PROGRAM MsgControl
VAR_INPUT
	TransmitEnable 				: BOOL;
	nConnectionIndex			: UDINT	:= 1;
END_VAR
VAR
	MsgID						: DINT;			// TCP/IP Message ID as per Communication protocol defined in FA 
	DeviceID					: STRING(5);	// TCP/IP Device ID as per Communication protocol defined in FA 
	BarCode						: STRING(20);	// TCP/IP Load ID (Bar Code) as per Communication protocol defined in FA
	BarCodeNoSpace				: STRING(20);	// TCP/IP Load ID (Bar Code) as per Communication protocol defined in FA stripped of spaces  
	Destination					: DINT;			// TCP/IP Destination as per Communication protocol defined in FA
	DefDestination				: DINT;			// TCP/IP Default Destination as per Communication protocol defined in FA
	Status						: BYTE;				// 
	Msg_EquipStatArry			: ARRAY[1..7] OF ST_Msg_EquipStat;
	nSystemStatusIndex 			: DINT; 	// Index used for Processing the system status array
	nTempOperState 				: DINT;	//Capture the Temporary Operating State of the Equipment for comparison
	nEquipStatusIndex			: DINT;	//Index used for adding items to the MSG_EquipStatArray
	StrStartPos					: INT;
	StrEndPos					: INT;
	MsgString					: STRING(55);
	RawMsgArray					: ARRAY[1..10] OF T_MaxString;	// Capture the last Raw messages for troubleshooting
	RawMsgLenArray				: ARRAY[1..10] OF INT;			// Capture the last  Raw message lengths for troubleshooting
	RawMsgStartPosArray			: ARRAY[1..10] OF INT;			// Capture the last  Raw message start positions for troubleshooting
	RawMsgEndPosArray			: ARRAY[1..10] OF INT;			// Capture the last  Raw message end positions for troubleshooting
	MsgArray					: ARRAY[1..10] OF STRING(55);		// Capture the last 10 messages that have been stripped from the starting character  for troubleshooting
	Blank_Msg_ConveyorStatArry	: ARRAY [1..7] OF ST_Msg_EquipStat := [7((Status := 99))];

	i 							: INT;
	j							: INT;
	
	RxCounter_Old				: UDINT;
	TxCounter_Old				: UDINT;
	TransmitMsgBuffer			: ARRAY [1..TransmitMsgBuffer_Size] OF STRING(55);	// Buffer to hold transmit messages
	TransmitMsgBuffer_Index		: INT :=	1;		// Index to the Buffer
	TransmitMsgStatus			: INT;			
	SendingMsg_Index			: INT :=	1;		// Index to send message
	
	ItemTransport				: ST_Item;		// Output Item Update with destination from ARUP Host (Send to Sorter PLC)
	BlankItem					: ST_Item := (ID := '', UniqueID := 0
													, Destination := 0
													, Status := E_StatusCode.No_Status
													, ExtStatus := E_StatusCode.No_Status
													, DeviceID := ''
													, MessageType := E_MessageIds.NoMessage_00);

	ReadBCRID_S2140_01_Old			: UDINT;		// Bar Code watch variable
	ReadBCRID_S2141_01_Old			: UDINT;		// Bar Code watch variable
	ReadBCRID_S2150_01_Old			: UDINT;		// Bar Code watch variable	
	ReadBCRID_S3080_01_Old			: UDINT;		// Bar Code watch variable
			
	TransmittedArray			: ARRAY[0..10] OF STRING(55);
	x							: DINT;
	y							: INT;
	
	SpacePosition				: INT;
	
	fb_CheckStopRegister		: FB_ManageCodes;	// Used to test for a specific Stop Code to report to the Host
	bOverHeight					: BOOL; 	// Detect OverHeight to report to the Host
	st_UpdateMessageToSend		: ST_Item;			// Message to Send to Host

	fb_SorterUpdateBuffer			: FB_ItemBuffer;	// Function to Process the SorterUpdateBuffer

	fb_SorterTransportBuffer_P2140	: FB_ItemBuffer;	// Function to Process the SorterTransportBuffer
	fb_SorterTransportBuffer_P2150	: FB_ItemBuffer;	// Function to Process the SorterTransportBuffer

	sMessage	:	STRING;
	
END_VAR

VAR CONSTANT
	SEND_ARRIVAL			:	INT := 5;
	SEND_LOCATION			:	INT := 7;
	TransmitMsgBuffer_Size	:	INT :=	25;		// Number of Messages to hold in buffer
END_VAR

// Create instances of Buffer Processing Functions to initialize the buffers and data
fb_SorterUpdateBuffer.Master := FALSE;
fb_SorterTransportBuffer_P2140.Master := TRUE;
fb_SorterTransportBuffer_P2150.Master := TRUE;

// Activate or de-activate logging
fb_SorterUpdateBuffer.LogEntries := .nItemBufferLogEnable.UPDATE OR .nItemBufferLogEnableP2150.UPDATE OR .nItemBufferLogEnableP2150.UPDATE;
fb_SorterTransportBuffer_P2140.LogEntries := .nItemBufferLogEnable.TRANSPORT OR .nItemBufferLogEnableP2140.TRANSPORT;
fb_SorterTransportBuffer_P2150.LogEntries := .nItemBufferLogEnable.TRANSPORT OR .nItemBufferLogEnableP2150.TRANSPORT;

// Setup Buffer names for Logging purposes
fb_SorterUpdateBuffer.Name := 'SYS UPDATE';
fb_SorterTransportBuffer_P2140.Name := 'P2140 SYS TRANSPORT';
fb_SorterTransportBuffer_P2150.Name := 'P2150 SYS TRANSPORT';

fb_SorterUpdateBuffer(st_BufferData := st_SorterUpdateBuffer
					, st_BufferFdbkIn := st_UpdateFdbkOut
					, st_BufferFdbkOut => st_UpdateFdbkIn);
fb_SorterTransportBuffer_P2140(st_BufferData := st_SorterTransportBuffer_P2140
					, st_BufferFdbkIn := st_TransportFdbkIn_P2140
					, st_BufferFdbkOut => st_TransportFdbkOut_P2140);
fb_SorterTransportBuffer_P2150(st_BufferData := st_SorterTransportBuffer_P2150
					, st_BufferFdbkIn := st_TransportFdbkIn_P2150
					, st_BufferFdbkOut => st_TransportFdbkOut_P2150);

(* -------------------- On Receive Message Process the data -------------------- *)
IF RxCounter_Old <> ServerControl.fbServer.aApplications[nConnectionIndex].RxCounter  THEN
	ItemTransport := BlankItem; // Clear the ItemTransport each pass to capture only new transport commands
	RECEIVE();
	// Test the DeviceID and route the Transport accordingly
	//	If there is only one possible DeviceID, this IF statement can be removed, but the fb_(TransportBuffer).AddItem call still has to be made
	//	Also, the default destination needs to be passed per DeviceID
	IF DeviceID = Sorter.st_Sorter_P2140Cfg.EquipID THEN
		// Added temporaily because code change needed on ARUP side 
			IF ItemTransport.Destination =0 THEN
			ItemTransport.Destination := 1;
			ELSIF ItemTransport.Destination =1 THEN
				ItemTransport.Destination := 2;
			END_IF
			// End addition	
		fb_SorterTransportBuffer_P2140.AddItem(st_ItemToAdd := ItemTransport);
		P2140_DefaultDestination := DefDestination;
	END_IF
	IF DeviceID = Sorter.st_Sorter_P2150Cfg.EquipID THEN
		fb_SorterTransportBuffer_P2150.AddItem(st_ItemToAdd := ItemTransport);
		P2150_DefaultDestination := DefDestination;
	END_IF

	RxCounter_Old := ServerControl.fbServer.aApplications[nConnectionIndex].RxCounter;
END_IF

(* -------------------- Transmit Messages if any are waiting in the buffer --------------------- *)
IF SendingMsg_Index <> TransmitMsgBuffer_Index THEN
	TRANSMIT(TransmitEnable:= TRUE);
END_IF

(* -------------------- Watch Bar code readers and send message when load is read -------------------- *)
(* ----- BCR_S2140_01: P2140 Divert  ----- *)	
ReadBCRID_S2140_01_Old := BarCodeMessage(cDatamanReader := BarCodeReaders.BCR_S2140_01
									, nOldCount := ReadBCRID_S2140_01_Old
									, nMessageToSend := SEND_ARRIVAL);
(* ----- BCR_S2141_01: P2143 Induct Confirm ----- *)	
ReadBCRID_S2141_01_Old := BarCodeMessage(cDatamanReader := BarCodeReaders.BCR_S2141_01
									, nOldCount := ReadBCRID_S2141_01_Old
									, nMessageToSend := SEND_LOCATION);
(* ----- BCR_S2150_01: P2150 Sorter ----- *)	
ReadBCRID_S2150_01_Old := BarCodeMessage(cDatamanReader := BarCodeReaders.BCR_S2150_01
									, nOldCount := ReadBCRID_S2150_01_Old
									, nMessageToSend := SEND_ARRIVAL);
(* ----- BCR_S3080_01: P3080 Lane Confirm ----- *)	
ReadBCRID_S3080_01_Old := BarCodeMessage(cDatamanReader := BarCodeReaders.BCR_S3080_01
									, nOldCount := ReadBCRID_S3080_01_Old
									, nMessageToSend := SEND_LOCATION);


(* -------------------- Watch Sorter and Device Status and transmit on change -------------------- *)
// Transmit On update from Sorter
// Detect a new message to process when the in and out pointer values disagree
IF st_SorterUpdateBuffer.nInPointer <> fb_SorterUpdateBuffer.OutPointer THEN
	// Pull the next message out of the buffer
	fb_SorterUpdateBuffer.RemoveItem(st_ItemToReturn => st_UpdateMessageToSend);
	CASE st_UpdateMessageToSend.MessageType OF

		E_MessageIds.TransportResponse_25:			// Response to a Transport Command

			CASE st_UpdateMessageToSend.Status OF
				E_StatusCode.Assign_Accepted:		// Assignment Accepted
					TransmitMsgStatus := E_TransportResponse.Accepted; 
				E_StatusCode.Assign_Full:			// Assigned Lane Unavailable
					TransmitMsgStatus := E_TransportResponse.DivertLaneUnavailable; 
				E_StatusCode.Assign_NotFound:		// Assigned Load ID Not Found
					TransmitMsgStatus := E_TransportResponse.LoadIdNotFound; 
				E_StatusCode.Assign_NotInducted:	// Assigned Load Not Inducted
					TransmitMsgStatus := E_TransportResponse.NextLoadReady; 
				E_StatusCode.Diverting:	// Assigned Load already Inducting
					TransmitMsgStatus := E_TransportResponse.LateInduction; 
			ELSE
				TransmitMsgStatus := E_TransportResponse.UnknownFailure; // Capture any other failures
				IF nMessageLogEnable.TransportResponse_25 THEN
					sMessage := CONCAT(' Item: ', st_UpdateMessageToSend.ID);
					sMessage := CONCAT(sMessage,' Destination: ');
					sMessage := CONCAT(sMessage, DINT_TO_STRING(st_UpdateMessageToSend.Destination));
					sMessage := CONCAT(sMessage,' TR Status: ');
					sMessage := CONCAT(sMessage, DINT_TO_STRING(st_UpdateMessageToSend.Status));
					// Write to the Error List
					ADSLOGSTR( msgCtrlMask := ADSLOG_MSGTYPE_HINT OR ADSLOG_MSGTYPE_LOG
						, msgFmtStr := 'Unhandled Transport Response Status: %s'
						, strArg := sMessage);
				END_IF
			END_CASE
			TransmitMsgBuffer[TransmitMsgBuffer_Index] := TransportResponse(Device := st_UpdateMessageToSend.DeviceID
																			, Barcode := st_UpdateMessageToSend.ID
																			, Status := TransmitMsgStatus);
			TransmitMsgBuffer_Index := IncIndex(TransmitMsgBuffer_Index,1,TransmitMsgBuffer_Size);

		E_MessageIds.TransportComplete_26:			// Indication of the final disposition of a transported item

			CASE st_UpdateMessageToSend.Status OF
				E_StatusCode.Divert_Success:		// Divert Success Message
					TransmitMsgStatus := E_TransportComplete.Success; 
				E_StatusCode.Divert_Complete:		// Divert Success Message
					TransmitMsgStatus := E_TransportComplete.Success; 
			ELSE 									// Catch all other failures
				TransmitMsgStatus := E_TransportComplete.Faulted; 
			END_CASE			
			CASE st_UpdateMessageToSend.ExtStatus OF
				E_StatusCode.Divert_Full:			// Divert Full/Unavailable
					TransmitMsgStatus := E_TransportComplete.Unavailable; 
				E_StatusCode.Divert_Offline:		// Divert Offline
					TransmitMsgStatus := E_TransportComplete.Offline; 
				E_StatusCode.Divert_Missed:		// Divert Missed
					TransmitMsgStatus := E_TransportComplete.Passed; 
				E_StatusCode.Divert_Recirculated:		// Divert Missed
					TransmitMsgStatus := E_TransportComplete.Success; 
			END_CASE			
			TransmitMsgBuffer[TransmitMsgBuffer_Index] := TransportComplete(Device:= st_UpdateMessageToSend.DeviceID
																			, BarCode:= st_UpdateMessageToSend.ID
																			, Dest:= DINT_TO_INT(st_UpdateMessageToSend.Destination)
																			, Status:= TransmitMsgStatus ); 
			TransmitMsgBuffer_Index := IncIndex(TransmitMsgBuffer_Index,1,TransmitMsgBuffer_Size);

	END_CASE
END_IF

// Transmit on Device Status Change
//DeviceStatus();1


(* -------------------- Reset The Transmit Triger after the message is succesfully added to the buffer ------------------- *)
IF ((ServerControl.fbServer.aApplications[nConnectionIndex].bTransmitTrigger = TRUE) OR ServerControl.TransmitTrigger = TRUE)  AND (TxCounter_Old <> ServerControl.fbServer.aApplications[nConnectionIndex].TxCounter) THEN
	ServerControl.TransmitTrigger := FALSE;
	TRANSMIT(TransmitEnable:= FALSE);
	TxCounter_Old := ServerControl.fbServer.aApplications[nConnectionIndex].TxCounter;
END_IF

METHOD PRIVATE Arrival : STRING(55)
VAR_INPUT
	Device :	STRING(5);		// Device Label per communication standard
	BarCode:	STRING(30);		// Barcode from barcode reader
	DefDest:	INT;		// Default destination
END_VAR
VAR
	String1: STRING(55);
	BC_Len: INT;
	x: INT;
	String_DefDest: STRING(2);
	y: INT;
	Device_Len: INT;
	i: INT;
END_VAR
(* Message from communication Spec:
	[STX (0x02h)][23][Device ID (5 CHR)][Barcode (20 CHR)][Default Dest (2 CHR)][Blank (22 CHR)][ETX 0x03h)]
*)

// Start Message with header
String1 := '$0223';

// Check Device for length and Pad with spaces if needed
Device_Len := LEN(Device);
IF Device_Len = 5 THEN
	String1 := CONCAT(STRING1, Device);
ELSIF Device_Len < 5 THEN
	String1 := CONCAT(STRING1, Device);
	FOR i := 1 TO (5-Device_Len) DO
		String1 := CONCAT(String1,' ');
	END_FOR
ELSE
	String1 := CONCAT(String1, 'XXXXX');
END_IF

// Check Barcode for length and Pad with spaces if needed
BC_Len := LEN(BARCODE);
IF BC_Len <20 THEN
	String1 := CONCAT(STRING1, BarCode);
	FOR x := 1 TO (20-BC_Len) DO
		String1 := CONCAT(String1,' ');
	END_FOR
ELSIF BC_Len = 20 THEN
	String1 := CONCAT(STRING1, BarCode);
ELSE 
	String1 := CONCAT(STRING1, RIGHT(BarCode,20));	
END_IF

// Check Default Destination for length and Pad with spaces if needed
String_DefDest := INT_TO_STRING(DefDest);
IF DefDest < 10 THEN
	String1 := CONCAT(String1,'0');
	String1 := CONCAT(String1, String_DefDest);
ELSIF (DefDest >= 10) AND (DefDest < 100) THEN
	String1 := CONCAT(String1, String_DefDest);
ELSE
	String1 := CONCAT(String1, 'XX');
END_IF	

// Pad with spaces
FOR y := 1 TO 22 DO
	String1 := CONCAT(String1,' ');
END_FOR

// Add ending Character
String1 := CONCAT(String1,'$03');
	
Arrival := String1;
END_METHOD

METHOD PRIVATE BarCodeMessage : UDINT
VAR_INPUT
	cDatamanReader	: CognexDataMan260;
//	sLocation		:	STRING(5);
	nOldCount		:	UDINT;
	nMessageToSend	: 	INT;
END_VAR
IF nOldCount <> cDatamanReader.GoodreadCount THEN
	// Send location update message to host
	CASE nMessageToSend OF
		SEND_ARRIVAL:	TransmitMsgBuffer[TransmitMsgBuffer_Index] := Arrival(cDatamanReader.In_EquipID, cDatamanReader.Out_ReadString,00);
		SEND_LOCATION: TransmitMsgBuffer[TransmitMsgBuffer_Index] := LocationUpdate(cDatamanReader.In_EquipID, cDatamanReader.Out_ReadString,00);
	END_CASE
	TransmitMsgBuffer_Index := IncIndex(TransmitMsgBuffer_Index,1,TransmitMsgBuffer_Size);
	BarCodeMessage := cDatamanReader.GoodreadCount;
ELSE
	BarCodeMessage := nOldCount;
END_IF
END_METHOD

METHOD PRIVATE CustomMessage : UDINT
VAR_INPUT
	EquipID			: 	STRING(5);
	Barcode			:	STRING(30);
	nReadCount		:	UDINT;
	nOldCount		:	UDINT;
	nMessageToSend	: 	INT;
END_VAR
IF nOldCount <> nReadCount THEN
	// Send location update message to host
	CASE nMessageToSend OF
		SEND_ARRIVAL:	TransmitMsgBuffer[TransmitMsgBuffer_Index] := Arrival(EquipID, BarCode,00);
		SEND_LOCATION: TransmitMsgBuffer[TransmitMsgBuffer_Index] := LocationUpdate(EquipID, BarCode,00);
	END_CASE
	TransmitMsgBuffer_Index := IncIndex(TransmitMsgBuffer_Index,1,TransmitMsgBuffer_Size);
	CustomMessage := nReadCount;
ELSE
	CustomMessage := nOldCount;
END_IF
END_METHOD

ACTION DeviceStatus:
(*
	
	Local Data items used for Equipment status processing
	Msg_EquipStatArry:	ARRAY[1..7] OF ST_Msg_EquipStat;
	nSystemStatusIndex : INT; 	// Index used for Processing the system status array
	nEquipStatusIndex: INT;	//Index used for adding items to the MSG_EquipStatArray
	nTempOperState : DINT;	//Capture the Temporary Operating State of the Equipment for comparison
	
	GVL_EquipmentArray items used for Equipment Status processing
	// System Equipment
	SystemEquip_Count : INT; //Count of Equipment to Process in System PLC
	SystemEquipStatusArray : ARRAY[1..EQUIP_COUNT_MAX] OF ST_StateCntrlSts; //Array of Equipment Status Current
	SystemEquipStatusArray_Last : ARRAY[1..EQUIP_COUNT_MAX] OF ST_StateCntrlSts; //Array of Equipment Status Last State
*)

//===================================================================================
(* 	Process the Conveyor/Equipment status arrays comparing the current state to the last state
 	When a state change is deteted, add the correspoding equipment to the Msg_EquipStatArray
		Then increment/test the nEquipStatusIndex and add the message to the outbound buffer
		if the Msg_EquipStatArry is full, and reset the nEquipStatusIndex value to the lower bound
*)
// Initialise the nEquipStatusIndex to 0 to detect when items are in the Msg_EquipStatArry buffer
nEquipStatusIndex := 0;

FOR nSystemStatusIndex := 1 TO gvl_equiparrays.nSystemEquip_Count BY 1 DO
	// Capture Offline State
	IF GVL_EquipArrays.aSystemEquipStatusArray[nSystemStatusIndex].CrntState = E_StateCntrl.stOffline THEN
		nTempOperState := E_EquipmentUpdate.Offline;
	ELSE
		// Capture Faulted State, or a specific Fault (in this instance, OverHeight)
		IF GVL_EquipArrays.aSystemEquipStatusArray[nSystemStatusIndex].CrntState = E_StateCntrl.stFaulted THEN
			// Check for an OverHeight in the Stop Register
			fb_CheckStopRegister.Check(nCodeToCheck := E_StopCodes.OverHeightFLT,
				bCodeSet => bOverHeight);
			// Set over Height
			IF bOverHeight THEN
				nTempOperState := E_EquipmentUpdate.OverHeight;
			ELSE
				// Otherwise, set Faulted
				nTempOperState := E_EquipmentUpdate.Faulted;
			END_IF
		ELSE
			// Capture Auto/Manual States and Running/Sleeping states where appropriate
			IF GVL_EquipArrays.aSystemEquipStatusArray[nSystemStatusIndex].CrntState = E_StateCntrl.stAuto THEN
				// Capture Auto-Running
				IF GVL_EquipArrays.aSystemEquipStatusArray[nSystemStatusIndex].CrntOperState = E_OperStateCntrl.running THEN
					nTempOperState := E_OperStateCntrl.running;
				// Capture Auto-Sleeping
				ELSIF GVL_EquipArrays.aSystemEquipStatusArray[nSystemStatusIndex].CrntOperState = E_OperStateCntrl.sleeping THEN
					nTempOperState := E_OperStateCntrl.sleeping;
				// Capture Auto
				ELSE
					nTempOperState := E_StateCntrl.stAuto;
				END_IF
			else
				// Capture Manual-Running
				IF GVL_EquipArrays.aSystemEquipStatusArray[nSystemStatusIndex].CrntOperState = E_OperStateCntrl.running THEN
					nTempOperState := E_OperStateCntrl.running;
				// Capture Manual
				ELSE
					nTempOperState := E_StateCntrl.stManual;
				END_IF
			end_if
		END_IF
	END_IF
	// Test for a change in Operatinal state or a non-initialized Storage array
	IF GVL_EquipArrays.aSystemEquipStatusArray_last[nSystemStatusIndex].LstOperState <> nTempOperState OR GVL_EquipArrays.aSystemEquipStatusArray_last[nSystemStatusIndex].Index = 0 THEN
		IF GVL_EquipArrays.aSystemEquipStatusArray_last[nSystemStatusIndex].Index = 0 THEN
			// Initialise the Storage Data Record
			GVL_EquipArrays.aSystemEquipStatusArray_last[nSystemStatusIndex] := GVL_EquipArrays.aSystemEquipStatusArray[nSystemStatusIndex];
		END_IF
		// Capture the nTempOperState for future comparisons
		GVL_EquipArrays.aSystemEquipStatusArray_last[nSystemStatusIndex].LstOperState := TO_INT(nTempOperState);
		// Increment the status index and check for roll-over
		nEquipStatusIndex := nEquipStatusIndex + 1;
		IF nEquipStatusIndex > 7 THEN
			// When there are 7 status updates, create the message
			TransmitMsgBuffer[TransmitMsgBuffer_Index] := EquipStatUpdate(Msg_EquipStatArry);
			// Increment the buffer index
			TransmitMsgBuffer_Index := IncIndex(TransmitMsgBuffer_Index,1,TransmitMsgBuffer_Size);
			// Set the index for the next message
			nEquipStatusIndex := 1;
		END_IF
		// Capture the Label and Index of the current Equipment status record
		Msg_EquipStatArry[nEquipStatusIndex].DeviceID := GVL_EquipArrays.aSystemEquipStatusArray[nSystemStatusIndex].Label;
		Msg_EquipStatArry[nEquipStatusIndex].Status := TO_INT(nTempOperState);
	END_IF
END_FOR

// Detect unsent items in the Msg_EquipStatArry buffer
IF nEquipStatusIndex > 0 THEN
	// Prepare the Equipment Status Message
	TransmitMsgBuffer[TransmitMsgBuffer_Index] := EquipStatUpdate(Msg_EquipStatArry);
	// Add the Equipment Status Message to the outbound buffer
	TransmitMsgBuffer_Index := IncIndex(TransmitMsgBuffer_Index,1,TransmitMsgBuffer_Size);
END_IF
END_ACTION

METHOD PRIVATE EquipStatUpdate : STRING(55)
VAR_IN_OUT
	Msg_ConveyorStatArry:	ARRAY[1..7] OF ST_Msg_EquipStat; // Array of Device status
END_VAR
VAR
	String1: STRING(55);
	x: INT;
	String_DefDest: STRING(2);
	y: INT;
	String_Status: STRING(2);
	Device_Len: INT;
	i: INT;
END_VAR
(* Message from communication Spec:
	[STX (0x02h)][28][Device 1 ID (5 CHR)][Status (2 CHR)] repeated for devices thru 7[ETX 0x03h)]
*)

// Start Message with header
String1 := '$0228';

FOR x := 1 TO 7 DO
	IF (Msg_ConveyorStatArry[x].DeviceID <> '') THEN
		// Check Device for length and Pad with spaces if needed
		Device_Len := LEN(Msg_ConveyorStatArry[x].DeviceID);
		IF Device_Len = 5 THEN
			String1 := CONCAT(String1,Msg_ConveyorStatArry[x].DeviceID);
		ELSIF Device_Len < 5 THEN
			Device_Len := LEN(Msg_ConveyorStatArry[x].DeviceID);
			FOR i := 1 TO (5-Device_Len) DO
				String1 := CONCAT(String1,' ');
			END_FOR
		ELSE
			String1 := CONCAT(String1, 'XXXXX');
		END_IF
		// Clear the DeviceID after processing
		Msg_ConveyorStatArry[x].DeviceID := '';
		
	
		// Check Status for length and Pad with spaces if needed
		String_Status := INT_TO_STRING(Msg_ConveyorStatArry[x].Status);
		IF Msg_ConveyorStatArry[x].Status < 10 THEN
			String1 := CONCAT(String1,'0');
			String1 := CONCAT(String1, String_Status);
		ELSIF (Msg_ConveyorStatArry[x].Status >= 10) AND (Msg_ConveyorStatArry[x].Status < 100) THEN
			String1 := CONCAT(String1, String_Status);
		ELSE
			String1 := CONCAT(String1, 'XX');
		END_IF	
		// Clear the Status after processing
		Msg_ConveyorStatArry[x].Status := 0;
	ELSE 
		String1 := CONCAT(String1,'       ');
	END_IF	
END_FOR

// Add ending Character
String1 := CONCAT(String1,'$03');
	
EquipStatUpdate := String1;
END_METHOD

METHOD PRIVATE KeepAliveResponse : STRING(55)
VAR_INPUT
END_VAR
VAR
	String1: STRING(55);
	x: INT;
END_VAR
(* Message from communication Spec:
	[STX (0x02h)][29][Blank (49 CHR)][ETX 0x03h)]
*)

// Start Message with header
String1 := '$0229';

// Pad with Spaces
FOR x := 1 TO 49 DO
	String1 := CONCAT(String1,' ');
END_FOR

// Add ending Character
String1 := CONCAT(String1,'$03');
	
KeepAliveResponse := String1;
END_METHOD

METHOD PRIVATE LocationUpdate : STRING(55)
VAR_INPUT
	Device :	STRING(5);		// Device Label per communication standard
	BarCode:	STRING(30);		// Barcode from barcode reader
	Dest:	INT;		// Default destination
END_VAR
VAR
	String1: STRING(55);
	BC_Len: INT;
	x: INT;
	String_Dest: STRING(2);
	y: INT;
	Device_Len: INT;
	i: INT;
END_VAR
(* Message from communication Spec:
	[STX (0x02h)][27][Device ID (5 CHR)][Barcode (20 CHR)][Destination (2 CHR)][Blank (24 CHR)][ETX 0x03h)]
*)

// Start Message with header
String1 := '$0227';

// Check Device for length and Pad with spaces if needed
Device_Len := LEN(Device);
IF Device_Len = 5 THEN
	String1 := CONCAT(STRING1, Device);
ELSIF Device_Len < 5 THEN
	String1 := CONCAT(STRING1, Device);
	FOR i := 1 TO (5-Device_Len) DO
		String1 := CONCAT(String1,' ');
	END_FOR	
ELSE
	String1 := CONCAT(String1, 'XXXXX');
END_IF


// Check Barcode for length and Pad with spaces if needed
BC_Len := LEN(BARCODE);
IF BC_Len <20 THEN
	String1 := CONCAT(STRING1, BarCode);
	FOR x := 1 TO (20-BC_Len) DO
		String1 := CONCAT(String1,' ');
	END_FOR
ELSIF BC_Len = 20 THEN
	String1 := CONCAT(STRING1, BarCode);
ELSE 
	String1 := CONCAT(STRING1, RIGHT(BarCode,20));	
END_IF

(* Destination isn't needed in location Update 
// Check Default Destination for length and Pad with spaces if needed
String_Dest := INT_TO_STRING(Dest);
IF Dest < 10 THEN
	String1 := CONCAT(String1,'0');
	String1 := CONCAT(String1, String_Dest);
ELSIF (Dest >= 10) AND (Dest < 100) THEN
	String1 := CONCAT(String1, String_Dest);
ELSE
	String1 := CONCAT(String1, 'XX');
END_IF	
*)

// Pad with spaces
FOR y := 1 TO 24 DO
	String1 := CONCAT(String1,' ');
END_FOR

// Add ending Character
String1 := CONCAT(String1,'$03');
	
LocationUpdate := String1;
END_METHOD

ACTION RECEIVE:
// Empty all outputs
	DeviceID := BarCode := '';
	Destination := DefDestination := 0;
	Status := 99;
	Msg_EquipStatArry := Blank_Msg_ConveyorStatArry;

	// Set up index with clipping to keep it within array boundaries	
	i := IncIndex(i,1,10);
		
	// Clear one before to make it easy to find newest entry 
	IF i = 10 THEN
		RawMsgArray[1] := '';	
		RawMsgLenArray[1] := 0;	
		RawMsgStartPosArray[1] := 0;
		RawMsgEndPosArray[1] :=  0;
	ELSE
		RawMsgArray[i+1] := '';	
		RawMsgLenArray[i+1] := 0;	
		RawMsgStartPosArray[i+1] := 0;
		RawMsgEndPosArray[i+1] :=  0;
	END_IF
	
	
	// Fill Appropriate info for each message
	RawMsgArray[i] := ServerControl.fbServer.aApplications[nConnectionIndex].RxRawMessage;	
	RawMsgLenArray[i] := LEN(ServerControl.fbServer.aApplications[nConnectionIndex].RxRawMessage);	
	StrStartPos := FIND(STR1:= RawMsgArray[i], STR2:='$02' );
	StrEndPos :=  FIND(STR1:= RawMsgArray[i], STR2:='$03' );
	RawMsgStartPosArray[i] := StrStartPos;
	RawMsgEndPosArray[i] := StrEndPos;
	
{info 'Maybe: Possibly add do while loop here to process the case where more than one message comes in at a time and clean up StrStartPos and end pos with array'}	
	IF StrStartPos <> 0 THEN
		MsgString := MID(STR:=ServerControl.fbServer.aApplications[nConnectionIndex].RxRawMessage , LEN:= 51 , POS:= StrStartPos);
		MsgArray[i] := MsgString;
		MsgID := STRING_TO_DINT(MID(STR:=ServerControl.fbServer.aApplications[nConnectionIndex].RxRawMessage , LEN:= 2, POS:= StrStartPos+1));
	
		CASE MsgID OF
			E_MessageIds.TransportCommand_05:  	// Transport Command Message
				DeviceID := MID(STR:=ServerControl.fbServer.aApplications[nConnectionIndex].RxRawMessage, LEN:= 5, POS:= StrStartPos+3);
				BarCode := MID(STR:=ServerControl.fbServer.aApplications[nConnectionIndex].RxRawMessage, LEN:= 20, POS:= StrStartPos+8);
				Destination := STRING_TO_DINT( MID(STR:=ServerControl.fbServer.aApplications[nConnectionIndex].RxRawMessage, LEN:= 2, POS:= StrStartPos+28));
				DefDestination := STRING_TO_DINT( MID(STR:=ServerControl.fbServer.aApplications[nConnectionIndex].RxRawMessage, LEN:= 2, POS:= StrStartPos+30));
				Status := STRING_TO_BYTE( MID(STR:=ServerControl.fbServer.aApplications[nConnectionIndex].RxRawMessage , LEN:= 2, POS:= StrStartPos+50));

				//Strip spaces from Bar Code
				SpacePosition := (FIND(STR1:= BarCode, STR2:=' ' ))+3;
				BarCodeNoSpace := MID(STR:=BarCode, LEN:= (20-SpacePosition), POS:= 1);
				// Update Info to send to Sorter PLC
//				ItemTransport := BlankItem;
				ItemTransport.DeviceID := DeviceID;
				ItemTransport.ID := BarCodeNoSpace;
				ItemTransport.Destination := Destination;
				ItemTransport.Status := E_StatusCode.UpdateNeeded;
				ItemTransport.MessageType := E_MessageIds.TransportCommand_05;
//				fb_SorterTransportBuffer.AddItem(st_ItemToAdd := ItemTransport);
//				Out_DefaultDestination := DefDestination;

			E_MessageIds.LocationUpdateResponse_07:		// Location Update Response
				DeviceID := MID(STR:=ServerControl.fbServer.aApplications[nConnectionIndex].RxRawMessage , LEN:= 5, POS:= StrStartPos+3);
				BarCode := MID(STR:=ServerControl.fbServer.aApplications[nConnectionIndex].RxRawMessage , LEN:= 20, POS:= StrStartPos+8);
				Destination := STRING_TO_DINT( MID(STR:=ServerControl.fbServer.aApplications[nConnectionIndex].RxRawMessage , LEN:= 2, POS:= StrStartPos+23));
				Status := STRING_TO_BYTE( MID(STR:=ServerControl.fbServer.aApplications[nConnectionIndex].RxRawMessage , LEN:= 2, POS:= StrStartPos+50));
						
			E_MessageIds.EquipmentStatusResponse_08:		// Equipment Status Response
				FOR j := 0 TO 6 DO
					Msg_EquipStatArry[j+1].DeviceID := MID(STR:=ServerControl.fbServer.aApplications[nConnectionIndex].RxRawMessage , LEN:= 5, POS:= ((StrStartPos+3)+(j*7)));
					Msg_EquipStatArry[j+1].Status := STRING_TO_BYTE(MID(STR:=ServerControl.fbServer.aApplications[nConnectionIndex].RxRawMessage , LEN:= 2, POS:= ((StrStartPos+8)+(j*7))));	
				END_FOR
			
			E_MessageIds.KeepAlive_09:		// Keep Alive
				// If Keep Alive message is recieved send the response to the transmit buffer
				TransmitMsgBuffer[TransmitMsgBuffer_Index] := KeepAliveResponse();
				TransmitMsgBuffer_Index := IncIndex(TransmitMsgBuffer_Index,1,TransmitMsgBuffer_Size);				
		END_CASE
	END_IF
END_ACTION

ACTION TRANSMIT:

// Transmit messages from buffer
IF NOT ServerControl.TransmitTrigger AND TransmitEnable THEN
	ServerControl.TxMessage := TransmitMsgBuffer[SendingMsg_Index];
	ServerControl.TransmitTrigger := TRUE;
	SendingMsg_Index := IncIndex(SendingMsg_Index,1,TransmitMsgBuffer_Size);
	
	TransmittedArray[y] := ServerControl.TxMessage;
	// Clear out message before last update to ease in testing
	IF y = 10 THEN
		TransmittedArray[1] := '';
	ELSE
		TransmittedArray[y+1] := '';
	END_IF
	
	y :=  IncIndex(IDX:= y, IdxMIN:= 0, IdxMAX:=10 );
END_IF
END_ACTION

METHOD PRIVATE TransportComplete : STRING(55)
VAR_INPUT
	Device :	STRING(5);		// Device Label per communication standard
	BarCode:	STRING(30);		// Barcode from barcode reader
	Dest:	INT;		// Default destination
	Status:	INT;		// Status
END_VAR
VAR
	String1: STRING(55);
	BC_Len: INT;
	x: INT;
	String_Dest: STRING(2);
	y: INT;
	String_Status: STRING(2);
	Device_Len: INT;
	i: INT;
END_VAR
(* Message from communication Spec:
	[STX (0x02h)][26][Device ID (5 CHR)][Barcode (20 CHR)][Destination (2 CHR)][Blank (20 CHR)][Status (2 CHR)][ETX 0x03h)]
*)

// Start Message with header
String1 := '$0226';

// Check Device for length and Pad with spaces if needed
Device_Len := LEN(Device);
IF Device_Len = 5 THEN
	String1 := CONCAT(STRING1, Device);
ELSIF Device_Len < 5 THEN
	String1 := CONCAT(STRING1, Device);
	FOR i := 1 TO (5-Device_Len) DO
		String1 := CONCAT(String1,' ');
	END_FOR
ELSE
	String1 := CONCAT(String1, 'XXXXX');
END_IF

// Check Barcode for length and Pad with spaces if needed
BC_Len := LEN(BARCODE);
IF BC_Len <20 THEN
	String1 := CONCAT(STRING1, BarCode);
	FOR x := 1 TO (20-BC_Len) DO
		String1 := CONCAT(String1,' ');
	END_FOR
ELSIF BC_Len = 20 THEN
	String1 := CONCAT(STRING1, BarCode);
ELSE 
	String1 := CONCAT(STRING1, RIGHT(BarCode,20));	
END_IF

// Check Destination for length and Pad with spaces if needed
String_Dest := INT_TO_STRING(Dest);
IF Dest < 10 THEN
	String1 := CONCAT(String1,'0');
	String1 := CONCAT(String1, String_Dest);
ELSIF (Dest >= 10) AND (Dest < 100) THEN
	String1 := CONCAT(String1, String_Dest);
ELSE
	String1 := CONCAT(String1, 'XX');
END_IF	

// Pad with Spaces
FOR y := 1 TO 20 DO
	String1 := CONCAT(String1,' ');
END_FOR

// Check Status for length and Pad with spaces if needed
String_Status := INT_TO_STRING(Status);
IF Status < 10 THEN
	String1 := CONCAT(String1,'0');
	String1 := CONCAT(String1, String_Status);
ELSIF (Status >= 10) AND (Status < 100) THEN
	String1 := CONCAT(String1, String_Status);
ELSE
	String1 := CONCAT(String1, 'XX');
END_IF	

// Add ending Character
String1 := CONCAT(String1,'$03');
	
TransportComplete := String1;
END_METHOD

METHOD PRIVATE TransportResponse : STRING(55)
VAR_INPUT
	Device :	STRING(5);		// Device Label per communication standard
	BarCode :	STRING(30);		// Barcode from barcode reader
	Status :	INT;		// Status
END_VAR
VAR
	String1: STRING(55);
	BC_Len: INT;
	x: INT;
	String_Status: STRING(2);
	y: INT;
	Device_Len: INT;
	i: INT;
END_VAR
(* Message from communication Spec:
	[STX (0x02h)][25][Device ID (5 CHR)][Barcode (20 CHR)][Blank (22 CHR)][Status (2 CHR)][ETX 0x03h)]
*)

// Start Message with header
String1 := '$0225';

// Check Device for length and Pad with spaces if needed
Device_Len := LEN(Device);
IF Device_Len = 5 THEN
	String1 := CONCAT(STRING1, Device);
ELSIF Device_Len < 5 THEN
	String1 := CONCAT(STRING1, Device);
	FOR i := 1 TO (5-Device_Len) DO
		String1 := CONCAT(String1,' ');
	END_FOR
ELSE
	String1 := CONCAT(String1, 'XXXXX');
END_IF

// Check Barcode for length and Pad with spaces if needed
BC_Len := LEN(BARCODE);
IF BC_Len <20 THEN
	String1 := CONCAT(STRING1, BarCode);
	FOR x := 1 TO (20-BC_Len) DO
		String1 := CONCAT(String1,' ');
	END_FOR
ELSIF BC_Len = 20 THEN
	String1 := CONCAT(STRING1, BarCode);
ELSE 
	String1 := CONCAT(STRING1, RIGHT(BarCode,20));	
END_IF

// Pad with Spaces
FOR y := 1 TO 22 DO
	String1 := CONCAT(String1,' ');
END_FOR

// Check Status for length and Pad with spaces if needed
String_Status := INT_TO_STRING(Status);
IF Status < 10 THEN
	String1 := CONCAT(String1,'0');
	String1 := CONCAT(String1, String_Status);
ELSIF (Status >= 10) AND (Status < 100) THEN
	String1 := CONCAT(String1, String_Status);
ELSE
	String1 := CONCAT(String1, 'XX');
END_IF

// Add ending Character
String1 := CONCAT(String1,'$03');
	
TransportResponse := String1;
END_METHOD

END_PROGRAM

(* stored: Version 1.1.0.1, ProductVersion 3.1.4024.4
   POU MsgControl: Id {2ad4410f-a5b6-449d-a112-8dab3c58adad}, SpecialFunc None
   Method Arrival: Id {393b8523-a43e-4b0d-b4b5-7c64712e9e9d}
   Method BarCodeMessage: Id {2d1b083e-f12e-4a46-aa5e-2e6d76ae375f}
   Method CustomMessage: Id {67e38799-204c-44b3-9a2f-aadccb796922}
   Action DeviceStatus: Id {6f2ea99a-b2ad-4c65-9c09-93cefc1dbe51}
   Method EquipStatUpdate: Id {2321939e-111c-4b05-8eb0-93df00614849}
   Method KeepAliveResponse: Id {84673126-43a8-4636-afc5-ab945f436879}
   Method LocationUpdate: Id {15f56496-1fb9-477c-86da-9bec7473c08d}
   Action RECEIVE: Id {e22fb3b2-e33a-4f01-9566-e2de5aea02ef}
   Action TRANSMIT: Id {a974ddda-c5af-4d9c-b0e3-1d4059ab2082}
   Method TransportComplete: Id {02cc8415-546f-4abe-b8b8-02bcdfae1f8d}
   Method TransportResponse: Id {e83eacf8-a434-47e5-8683-cc87bbe6c34d} *)
